Staubli VAL3: onLeftEvent.pgx

program onLeftEvent()
begin
  call save:BackBoxType()
  call buildList()
end
